FUNCTION_BLOCK IO_DI32_HMI (* Service Interface Function Block Type *)
  (* Standard: 61499-2 *)
  (* Version 0.0, 10/2/2026, Schneider Electric, template *)
  PACKAGE Hidryco.HidrycoLib;
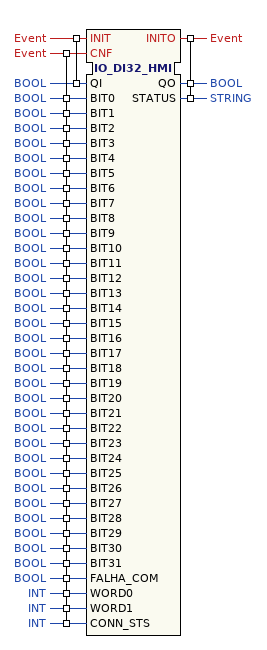
  EVENT_INPUT
    INIT WITH QI;
    CNF WITH BIT0, BIT1, BIT2, BIT3, BIT4, BIT5, BIT6, BIT7, BIT8, BIT9, BIT10, BIT11, BIT12, BIT13, BIT14, BIT15, BIT16, BIT17, BIT18, BIT19, BIT20, BIT21, BIT22, BIT23, BIT24, BIT25, BIT26, BIT27, BIT28, BIT29, BIT30, BIT31, FALHA_COM, WORD0, WORD1, CONN_STS; (* Atualiza o depurador *)
  END_EVENT
  EVENT_OUTPUT
    INITO WITH QO, STATUS;
  END_EVENT
  VAR_INPUT
    QI : BOOL;
    BIT0 : BOOL; (* DI 0 *)
    BIT1 : BOOL; (* DI 1 *)
    BIT2 : BOOL; (* DI 2 *)
    BIT3 : BOOL; (* DI 3 *)
    BIT4 : BOOL; (* DI 4 *)
    BIT5 : BOOL; (* DI 5 *)
    BIT6 : BOOL; (* DI 6 *)
    BIT7 : BOOL; (* DI 7 *)
    BIT8 : BOOL; (* DI 8 *)
    BIT9 : BOOL; (* DI 9 *)
    BIT10 : BOOL; (* DI 10 *)
    BIT11 : BOOL; (* DI 11 *)
    BIT12 : BOOL; (* DI 12 *)
    BIT13 : BOOL; (* DI 13 *)
    BIT14 : BOOL; (* DI 14 *)
    BIT15 : BOOL; (* DI 15 *)
    BIT16 : BOOL; (* DI 16 *)
    BIT17 : BOOL; (* DI 17 *)
    BIT18 : BOOL; (* DI 18 *)
    BIT19 : BOOL; (* DI 19 *)
    BIT20 : BOOL; (* DI 20 *)
    BIT21 : BOOL; (* DI 21 *)
    BIT22 : BOOL; (* DI 22 *)
    BIT23 : BOOL; (* DI 23 *)
    BIT24 : BOOL; (* DI 24 *)
    BIT25 : BOOL; (* DI 25 *)
    BIT26 : BOOL; (* DI 26 *)
    BIT27 : BOOL; (* DI 27 *)
    BIT28 : BOOL; (* DI 28 *)
    BIT29 : BOOL; (* DI 29 *)
    BIT30 : BOOL; (* DI 30 *)
    BIT31 : BOOL; (* DI 31 *)
    FALHA_COM : BOOL; (* TRUE = remota offline *)
    WORD0 : INT; (* Word 0 (bits 0-15) *)
    WORD1 : INT; (* Word 1 (bits 16-31) *)
    CONN_STS : INT; (* connStatusInt: 1 online, 0 offline *)
  END_VAR
  VAR_OUTPUT
    QO : BOOL; (* Event Output Qualifier *)
    STATUS : STRING; (* Service Status *)
  END_VAR
  SERVICE /
    SEQUENCE 
    END_SEQUENCE
  END_SERVICE
END_FUNCTION_BLOCK
